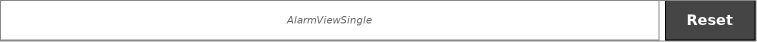
VISUALIZATION AlarmViewSingleWithReset  // 757x42
VAR_IN_OUT
  reset: BOOL;
END_VAR
VAR_INPUT
  event_message: EventMessageHMI;
  forward_visu: STRING;
END_VAR
    Frame (0,0 659x40)
        shows AlarmViewSingle(event_message := event_message)
        OnMouseClick: change screen: AssignExpression forward_visu
    Rectangle (665,0 90x40), "Reset"
        tap reset
END_VISUALIZATION

(* stored: Version 1.1.0.1, ProductVersion 3.1.4022.18
   Visu AlarmViewSingleWithReset: Id {911b0036-64ca-430b-935a-661773d7d46a} *)
